FUNCTION_BLOCK E_RESTART (* Generation of Restart Events *)
  (* Standard: 61499-1-A.1; Description: Generation of restart events *)
  (* Version 0.0, 2001-03-25, JHC, Rockwell Automation, First XML version. *)
  (* Compiler header: package fb.rt.events; *)
  (* Compiler Java IBM VisualAge 3.0 *)
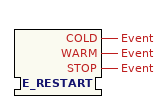
  EVENT_OUTPUT
    COLD; (* Cold Restart *)
    WARM; (* Warm Restart *)
    STOP; (* Resource is Stopping *)
  END_EVENT
  SERVICE RESOURCE/E_RESTART
    SEQUENCE cold_restart
      RESOURCE.start() -> E_RESTART.COLD();
    END_SEQUENCE
    SEQUENCE warm_restart
      RESOURCE.restart() -> E_RESTART.WARM();
    END_SEQUENCE
    SEQUENCE stopping
      RESOURCE.stop() -> E_RESTART.STOP();
    END_SEQUENCE
  END_SERVICE
END_FUNCTION_BLOCK
